// Usage:
// Call instance (i.e. ofbCsvRead();) every scan while waiting for operations to complete.
// SetFileParams() Set the File directory and separator variable. 
// GetFile() Get the File.
// #various props: Observe the properties to see whether it passed the file checks.
// NextField() Next through the fields of the CSV. 
// #sField, Row, Column: Use properties to access values, using row and column.
FUNCTION_BLOCK T_CsvFileReader
VAR
// state vars.
	filePath : Tc2_Utilities.T_MaxString; // filepath
	firstField : BOOL;
	newRow : BOOL;
	
// backing properties	
	_Row : UINT;(* Row number (record) *)
	_Column : UINT;(* Column number (record field) *)
	_Field : Tc2_Utilities.T_MaxString; // Field in current Row and column
	
// Objects	
	fileRead : T_FileReadBase;(* Writes one record (line) *)
	csvReader : Tc2_Utilities.FB_CSVMemBufferReader; // read bits
	
END_VAR

fileRead();

{attribute 'monitoring' := 'call'}
PROPERTY PUBLIC Busy : BOOL
GET
Busy := fileRead.Busy;
END_GET
END_PROPERTY

PROPERTY PUBLIC Column : UINT
GET
Column := _Column;
END_GET
END_PROPERTY

{attribute 'monitoring' := 'call'}
PROPERTY PUBLIC Eof : BOOL
GET
Eof := ReadyForParsing AND NOT csvReader.bOk AND NOT firstField;
END_GET
END_PROPERTY

{attribute 'monitoring' := 'call'}
PROPERTY PUBLIC Error : BOOL
GET
Error := fileRead.Error;
END_GET
END_PROPERTY

{attribute 'monitoring' := 'call'}
PROPERTY PUBLIC ErrorId : UDINT
GET
ErrorId := fileRead.ErrorId;
END_GET
END_PROPERTY

PROPERTY PUBLIC Field : String
GET
Field := _Field;
END_GET
END_PROPERTY

PROPERTY PUBLIC FileExists : BOOL
GET
FileExists := fileRead.FileExists;
END_GET
END_PROPERTY

METHOD PUBLIC GetFile
fileRead.StartRead();
fileRead();
_Column := 0;
_Row := 0;
_Field := '';
firstField := TRUE;
newRow := FALSE;
END_METHOD

METHOD PRIVATE incrementRowAndColumn
IF newRow THEN // if it's a new row (which we know from last time)
	
	newRow := FALSE;
	_Row := _Row + 1;
	_Column := 0;
	
ELSE
	// if it's not the first read, advance column.
	IF (csvReader.eCmd = Tc2_Utilities.eEnumCmd_First) THEN
		_Column := 0;
		_Row := 0;
	ELSE
		_Column := _Column + 1;
	END_IF
	
END_IF
END_METHOD

METHOD PUBLIC NextField// gets next field
IF firstField THEN
	firstField := FALSE;
	csvReader.eCmd :=  Tc2_Utilities.E_EnumCmdType.eEnumCmd_First;
ELSE
	csvReader.eCmd :=  Tc2_Utilities.E_EnumCmdType.eEnumCmd_Next;
END_IF

processCsvReader();

// increment the column and row if necessary.
IF csvReader.bOk THEN
	incrementRowAndColumn();
	
END_IF

// increment the row number next call if necessary.
IF csvReader.bOk AND csvReader.bCRLF THEN
	newRow := TRUE;
END_IF
END_METHOD

METHOD PRIVATE processCsvReader 
// used in NextField();
csvReader(
	pBuffer:= fileRead.DataBuffer,
	cbBuffer:= fileRead.DataLength,
	getValue=> _Field);
END_METHOD

{attribute 'monitoring' := 'call'}
PROPERTY PUBLIC ReadyForParsing : BOOL
GET
ReadyForParsing := fileRead.Done;
END_GET
END_PROPERTY

PROPERTY PUBLIC Row : UINT
GET
Row := _Row;
END_GET
END_PROPERTY

METHOD PUBLIC SetFileParams
VAR_INPUT
	FilePath : Tc2_Utilities.T_MaxString;
	Separator: BYTE; // Updates TC Utilities Global_Variables DEFAULT_CSV_FIELD_SEP
END_VAR
// THIS^ references the base object properties
THIS^.filePath := FilePath; // for debug only.

fileRead.SetFilePath(FilePath := FilePath);

// Validate separator.
IF Separator = ASCI_SEMI_COLON THEN
	Tc2_Utilities.DEFAULT_CSV_FIELD_SEP := 16#3B;
	
ELSIF Separator = ASCI_COMMA THEN
	Tc2_Utilities.DEFAULT_CSV_FIELD_SEP := 16#3B;
	
ELSE
	Tc2_Utilities.DEFAULT_CSV_FIELD_SEP := 16#3B;
	
END_IF
END_METHOD

END_FUNCTION_BLOCK

(* stored: Version 1.1.0.1, ProductVersion 3.1.4022.12
   POU T_CsvFileReader: Id {f698c541-82b7-49fe-a39a-d5b39221df43}, SpecialFunc None
   Folder Methods: Id {0ccf71fb-eff4-4971-bebb-f2db3f398075}
   Folder Privates: Id {c264b212-188f-492b-9d5d-cc8abd3f2e89}
   Folder Properties: Id {4d45de3b-a9fa-49c7-9cb2-a92c347c29b6}
   Property Busy: Id {e9ea1e4b-cede-4293-886f-61f164db727b}
   Get Get: Id {57989dfa-9851-4490-aa99-6e15ec5883fd}
   Property Column: Id {ca30f05a-c748-4363-9377-6e46d303b8de}
   Get Get: Id {549f03d3-34ec-453d-b404-8330c5f2ac87}
   Property Eof: Id {737915ef-d04e-4ef5-8e6f-d5be621f917c}
   Get Get: Id {a4c0e73e-a9aa-414b-a4e3-63b970de6ef0}
   Property Error: Id {2b039a65-a40a-45e9-b0b5-d2b67227bfba}
   Get Get: Id {5c6173da-7291-4db9-b693-dc6cfd4bca7a}
   Property ErrorId: Id {2f840b8b-6912-428f-8ae7-cf7a7bee0a56}
   Get Get: Id {e673318a-731c-4c2f-8177-20878d2a114a}
   Property Field: Id {865fbe2a-be60-4449-8c53-c3605f20d429}
   Get Get: Id {379e603a-abf4-4f3a-9b63-65a352852a0a}
   Property FileExists: Id {ad4c90e6-6627-49b1-a78e-459af2bf1656}
   Get Get: Id {72b8f14d-75ba-47fa-b5bb-69df465c867b}
   Method GetFile: Id {0079e725-90d6-42fd-b668-4fea4a4f856b}
   Method incrementRowAndColumn: Id {cf7aeecd-725d-46ac-bab5-43ab50603bc3}
   Method NextField: Id {2069769d-95b0-4488-94ec-06795445d487}
   Method processCsvReader: Id {19f24496-c709-448c-9747-2fc3b8ae16d2}
   Property ReadyForParsing: Id {6ac0ed30-b635-4e9e-8e69-3853e7ad9f06}
   Get Get: Id {e158f41a-26cd-4222-a0f8-5f6c09312497}
   Property Row: Id {9c5a1564-789d-4eab-b829-6776c9f8ba8a}
   Get Get: Id {a52f8176-f083-4b67-be53-4cd001530fae}
   Method SetFileParams: Id {71df841a-242a-470f-b9d8-966ebc5a9863} *)
